FUNCTION_BLOCK FLOAT_TO_VECTOR_Z (* Creates a zero vector with z yielding the input float *)
  (* Standard: 61499-2 *)
  (* Version 1.0, 29-03-12, GASR, Universidade do Estado de Santa Catarina *)
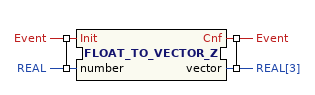
  EVENT_INPUT
    Init WITH number;
  END_EVENT
  EVENT_OUTPUT
    Cnf WITH vector;
  END_EVENT
  VAR_INPUT
    number : REAL;
  END_VAR
  VAR_OUTPUT
    vector : ARRAY [0..2] OF REAL;
  END_VAR
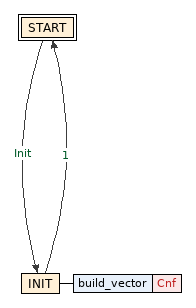
  EC_STATES
    START;
    INIT : build_vector -> Cnf;
  END_STATES
  EC_TRANSITIONS
    START TO INIT := Init;
    INIT TO START := 1;
  END_TRANSITIONS
  ALGORITHM build_vector IN Lua:
vector[1] = 0
vector[2] = 0
vector[3] = number
  END_ALGORITHM
END_FUNCTION_BLOCK
